// TIA Portal V17 export
// export: Created 2023-12-22T15:05:34.7775916Z, ExportSetting WithDefaults, DisplayName Totally Integrated Automation Portal, DisplayVersion V17, DisplayName TIA Portal Openness, DisplayVersion V17, DisplayName TIA Portal Version Control Interface, DisplayVersion V17, DisplayName STEP 7 Professional, DisplayVersion V17, DisplayName STEP 7 Safety, DisplayVersion V17, DisplayName WinCC Advanced, DisplayVersion V17
DATA_BLOCK "Comm_Scada"   // DB10
{ S7_Optimized_Access := 'FALSE' }
VERSION : 0.1
// stored: AutoNumber false, DBAccessibleFromOPCUA true, IsOnlyStoredInLoadMemory false, IsWriteProtectedInAS false
   VAR
      Input : Struct
         DI_AllBlock : Bool;   // Аварийный останов
         DI_EZ_1_FB_AHLS : Bool;   // Электролизер 1 (Переполнение поддона)
         DI_Gas_Chanel_1_1 : Bool;   // Загазованность канал 1 (Порог 1)
         DI_Gas_Chanel_1_2 : Bool;   // Загазованность канал 1 (Порог 2)
         DI_Gas_Chanel_2_1 : Bool;   // Загазованность канал 2 (Порог 1)
         DI_Gas_Chanel_2_2 : Bool;   // Загазованность канал 2 (Порог 2)
         DI_ALS_1 : Bool;   // Аварийный уровень 1
         ELZ_Wash : Bool;   // Идет промывка
         KC_1 : Bool;   // Промывка фильтра 1
         KC_2 : Bool;   // Промывка фильтра 2
         ELZ_Local : Bool;
         ELZ_1_Status : Int;   // Статус электролизера
         Pump_1_Status : Int;   // Статус насоса 1
         Pump_2_Status : Int;   // Статус насоса 2
         Pump_ELZ_Status : Int;   // Статус насоса электролизера
         RM_1 : Real;   // Импульсный расходомер
         Line_1_Flow_1 : Real;   // Дозирование гипохлорита линии 1
         Line_2_Flow_1 : Real;   // Дозирование гипохлорита линии 2
         AI_LE_1_Result : Real;   // Датчик уровня
         AI_TE_1_Result : Real;   // Датчик температуры
         ELZ_1_Alarm : Word;   // Слово аварий электролизера
         Pump_1_Alarm : Word;   // Слово аварий насоса 1
         Pump_2_Alarm : Word;   // Слово аварий насоса 2
         Pump_ELZ_Alarm : Word;   // Слово аварий электролизера
         AI_LE_1_Alarm : Word;   // Слово аварий датчика уровня
         AI_TE_1_Alarm : Word;   // Слово аварий датчика температуры
         Logick_Alarm : Word;   // Слово аварий блока логики
      END_STRUCT;
      Output : Struct
         Start_ELZ : Bool;   // Запуск электролизера
         Line_1_Start : Bool;   // Старт линии 1
         Line_2_Start : Bool;   // Старт линии 2
         Line_1_Flow : Real;   // Дозирование гипохлорита линии 1
         Line_2_Flow : Real;   // Дозирование гипохлорита линии 2
      END_STRUCT;
   END_VAR
BEGIN
END_DATA_BLOCK
